// TIA Portal V20 export
DATA_BLOCK "BK22"   // DB274
// stored: MemoryReserve 100
   VAR
      "X10-1.SEPA GRIPPER CLAMP OPEN" : Bool := TRUE;
      "X11-1.SPARE" : Bool := FALSE;
      "X12-1.SEPA GRIPPER CLAMP DETECT SENSOR" : Bool := TRUE;
      "X13-1.SEPA GRIPPER BACKWARD" : Bool := FALSE;
      "X14-1.SEPA GRIPPER C-AXIS LIMIT SENSOR(-)" : Bool := TRUE;
      "X15-1.SEPA GRIPPER C-AXIS LIMIT SENSOR(+)" : Bool := TRUE;
      "X16-1.SEPA GRIPPER Z-AXIS LIMIT SENSOR(-)" : Bool := TRUE;
      "X17-1.SEPA GRIPPER Z-AXIS LIMIT SENSOR(+)" : Bool := TRUE;
      "X10-2.SEPA GRIPPER CLAMP CLOSE" : Bool := FALSE;
      "X11-2.SPARE" : Bool := FALSE;
      "X12-2.SPARE" : Bool := FALSE;
      "X13-2.SEPA GRIPPER FORWARD" : Bool := FALSE;
      "X14-2.SEPA GRIPPER C-AXIS HOME SENSOR" : Bool := TRUE;
      "X15-2.SPARE" : Bool := FALSE;
      "X16-2.SEPA GRIPPER Z-AXIS HOME SENSOR" : Bool := TRUE;
      "X17-2.SPARE" : Bool := FALSE;
   END_VAR
BEGIN
END_DATA_BLOCK
